Staubli VAL3: sendStatus.pgx

program sendStatus()
begin
  for stringLen=0 to 15
    message2ASCII[stringLen]=asc(mid(message,1,stringLen),0)
  endFor
  sioSet(sioASCII,message2ASCII)
  delay(1)
end
